TYPE U_AXIS_MOVE_DATA :
UNION

  stCtrl              : ARRAY[1..MAX_AXIS] OF ST_AXIS_MOVE_DATA;

  byCtrl    AT %I*    : ARRAY[1..MAX_AXIS] OF
                        ARRAY[1..SIZEOF(ST_AXIS_MOVE_DATA)] OF BYTE;
END_UNION
END_TYPE

(* stored: Version 1.1.0.1, ProductVersion 3.1.4026.19
   DUT U_AXIS_MOVE_DATA: Id {e2995197-d128-089f-00b0-eef4250b8a19} *)
